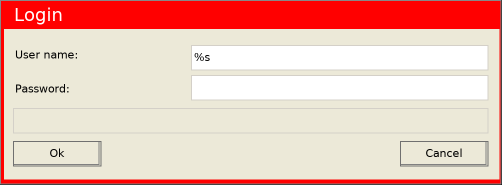
VISUALIZATION CustomLoginDialog  // 502x185
VAR
	iIndexLoginProvider : DWORD;
END_VAR
    Rectangle (0,0 502x185)
    Rectangle (4,29 495x150)
    Rectangle (11,0 476x30), "Login"
    Label (12,40 180x30), "User name:"
    Label (12,74 180x30), "Password:"
    Textfield (191,45 297x25), "%s", text variable: VisuUserManagement.g_VisuLoginProviderManager.m_arrLoginProvider[iIndexLoginProvider].stUserName
        OnMouseDown: write the text variable via Default
    Textfield (191,75 297x25), text variable: VisuUserManagement.g_VisuLoginProviderManager.m_arrLoginProvider[iIndexLoginProvider].stPassword
        OnMouseDown: write the text variable via Default, password
    Textfield (13,108 475x25), text list: '.VisuUserManagement.TL_VUM_Errors', text index: VisuUserManagement.g_VisuLoginProviderManager.m_arrLoginProvider[iIndexLoginProvider].udiLastError
    Button (13,141 88x25), "Ok"
        OnMouseDown: execute { VisuUserManagement.g_VisuLoginProviderManager.m_arrLoginProvider[iIndexLoginProvider].dwDialogResultOK := TRUE; }
    Button (400,141 88x25), "Cancel"
        OnMouseDown: execute { VisuUserManagement.g_VisuLoginProviderManager.m_arrLoginProvider[iIndexLoginProvider].dwDialogResultCancel := TRUE; }
END_VISUALIZATION

(* stored: Version 1.1.0.1, ProductVersion 3.1.4024.3
   Visu CustomLoginDialog: Id {c85f390c-d0e1-490f-9c5e-e9445bd87574} *)
